FUNCTION_BLOCK Organization (* Composite Function Block Type *)
  (* Standard: 61499-2 *)
  (* Version 0.0, 15/09/2021, Pranay Jhunjhunwala, Schneider Electric, template *)
  PACKAGE Main;
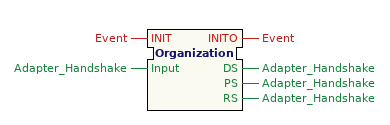
  EVENT_INPUT
    INIT; (* Initialization Request *)
  END_EVENT
  EVENT_OUTPUT
    INITO; (* Initialization Confirm *)
  END_EVENT
  SOCKETS
    Input : Adapter_Handshake;
  END_SOCKETS
  PLUGS
    DS : Adapter_Handshake;
    PS : Adapter_Handshake;
    RS : Adapter_Handshake;
  END_PLUGS
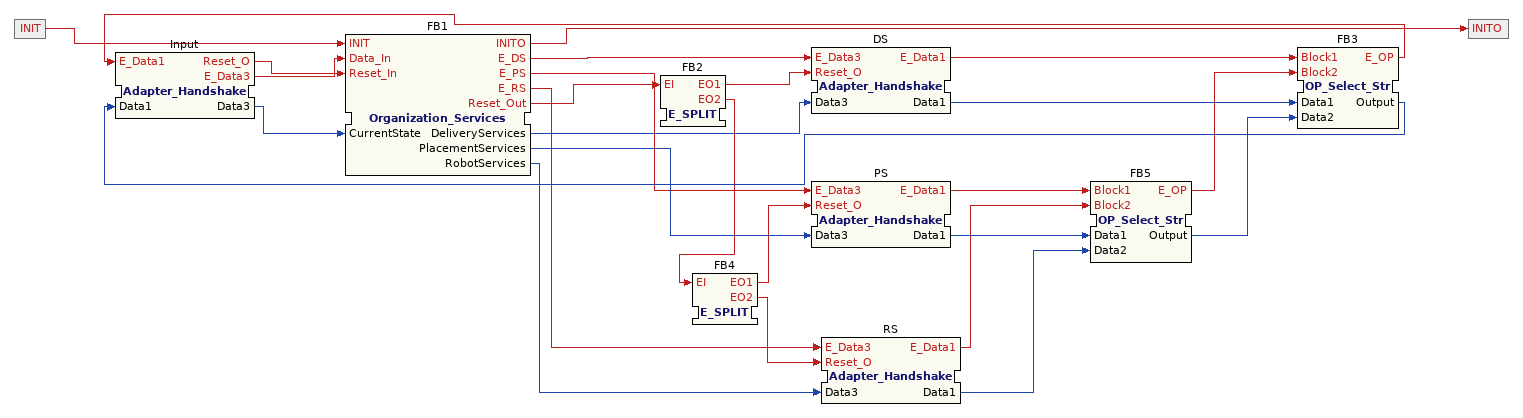
  FBS
    FB1 : Organization_Services;
    FB2 : E_SPLIT;
    FB3 : OP_Select_Str;
    FB4 : E_SPLIT;
    FB5 : OP_Select_Str;
  END_FBS
  EVENT_CONNECTIONS
    Input.Reset_O TO FB1.Reset_In;
    Input.E_Data3 TO FB1.Data_In;
    INIT TO FB1.INIT;
    FB1.INITO TO INITO;
    FB1.Reset_Out TO FB2.EI;
    FB1.E_PS TO PS.E_Data3;
    FB1.E_DS TO DS.E_Data3;
    FB2.EO1 TO DS.Reset_O;
    FB2.EO2 TO FB4.EI;
    DS.E_Data1 TO FB3.Block1;
    PS.E_Data1 TO FB5.Block1;
    FB3.E_OP TO Input.E_Data1;
    FB1.E_RS TO RS.E_Data3;
    FB4.EO1 TO PS.Reset_O;
    FB4.EO2 TO RS.Reset_O;
    RS.E_Data1 TO FB5.Block2;
    FB5.E_OP TO FB3.Block2;
  END_CONNECTIONS
  DATA_CONNECTIONS
    Input.Data3 TO FB1.CurrentState;
    FB1.DeliveryServices TO DS.Data3;
    FB1.PlacementServices TO PS.Data3;
    DS.Data1 TO FB3.Data1;
    PS.Data1 TO FB5.Data1;
    FB3.Output TO Input.Data1;
    FB1.RobotServices TO RS.Data3;
    RS.Data1 TO FB5.Data2;
    FB5.Output TO FB3.Data2;
  END_CONNECTIONS
END_FUNCTION_BLOCK
